(* Logix 5000 project; controller EuniceF_ICA20 vendor 1 type 14 code 150 rev 37.11; software revision 37.00 *)

TASK MainTask (continuous, watchdog 500 ms) : MainProgram

MODULES
   Local : vendor 1 type 14 code 150 (Compact 0, rev 37.11)
      Discrete_IO : Embedded (Compact 1, rev 3.1, Output RPI 20 ms)
      Analog_IO : Embedded (Compact 2, rev 1.1, Output RPI 80 ms)
      Counters : Embedded (Compact 3, rev 1.1, Output RPI 20 ms)
END_MODULES

VAR_GLOBAL   (* controller tags *)
   AI_Voltage_Raw : ALIAS FOR Local:2:I.Ch0Data;
   Current : REAL;
   current_mess : STRING;
   current_per : STRING;
   Current_Raw : ALIAS FOR Local:2:I.Ch1Data;
   Main_message : STRING;
   PercentCurrent : REAL;
   PercentVoltage : REAL;
   Switch : ALIAS FOR Local:1:I.Data.1;
   Temp_Current : STRING;
   Temp_perCurrent : STRING;
   Temp_perVoltage : STRING;
   Temp_Voltage : STRING;
   Txt_Current : STRING := 'The Current is: ';
   Txt_mA : STRING := ' mA| ';
   Txt_Percent : STRING := ' %';
   Txt_V : STRING := ' mV| ';
   Txt_Voltage : STRING := 'The voltage is : ';
   Voltage : REAL;
   voltage_mess : STRING;
   voltage_per : STRING;
END_VAR

PROGRAM MainProgram   (* main routine MainRoutine *)

ROUTINE MainRoutine   (* ladder *)
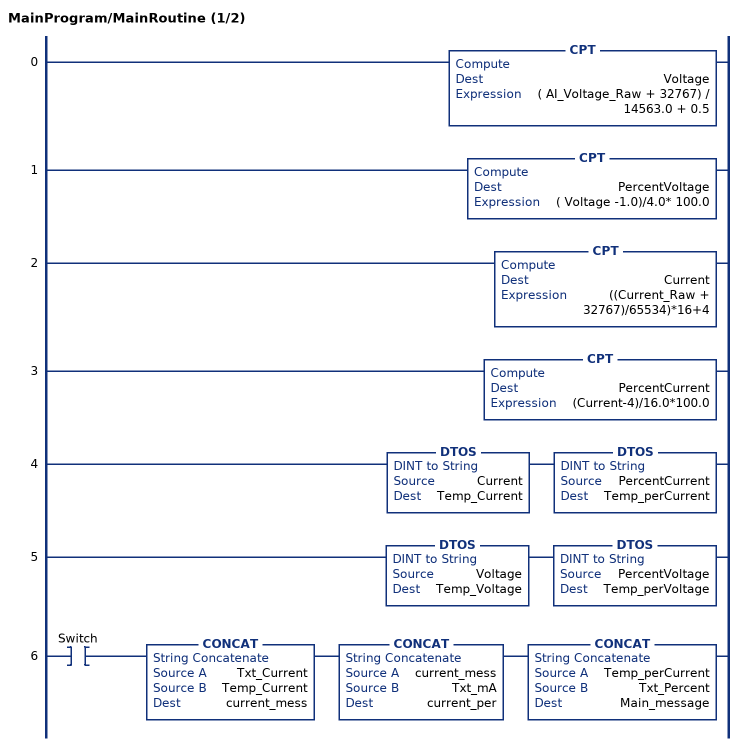
   0: CPT(Voltage,( AI_Voltage_Raw + 32767) / 14563.0 + 0.5);
   1: CPT(PercentVoltage,( Voltage -1.0)/4.0* 100.0);
   2: CPT(Current,((Current_Raw + 32767)/65534)*16+4);
   3: CPT(PercentCurrent,(Current-4)/16.0*100.0);
   4: DTOS(Current,Temp_Current)DTOS(PercentCurrent,Temp_perCurrent);
   5: DTOS(Voltage,Temp_Voltage)DTOS(PercentVoltage,Temp_perVoltage);
   6: XIC(Switch)CONCAT(Txt_Current,Temp_Current,current_mess)CONCAT(current_mess,Txt_mA,current_per)CONCAT(Temp_perCurrent,Txt_Percent,Main_message);
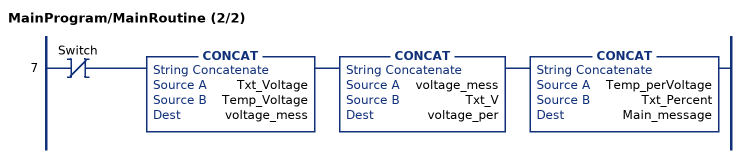
   7: XIO(Switch)CONCAT(Txt_Voltage,Temp_Voltage,voltage_mess)CONCAT(voltage_mess,Txt_V,voltage_per)CONCAT(Temp_perVoltage,Txt_Percent,Main_message);
END_ROUTINE
END_PROGRAM
